TYPE ST_BottleTypeParams :
STRUCT
	stLoadingBottleParams:ST_LoadingBottleParams;
	stWeighingBottleParams:ST_WeighingBottleParams;
	stUnloadingBottleParams:ST_UnloadingBottleParams;
END_STRUCT
END_TYPE

(* stored: Version 1.1.0.1, ProductVersion 3.1.4024.15
   DUT ST_BottleTypeParams: Id {9d0e5e67-e809-4ee8-abd1-9105770df435} *)
